// TIA Portal V20 export
// export: Created 2025-12-01T14:57:05.3623851Z, ExportSetting None, DisplayName Totally Integrated Automation Portal, DisplayVersion V20 Update 3, DisplayName TIA Portal Openness, DisplayVersion V20 Update 3, DisplayName TIA Portal Version Control Interface, DisplayVersion V20 Update 3, DisplayName STEP 7 Professional, DisplayVersion V20 Update 3, DisplayName STEP 7 Safety, DisplayVersion V20 Update 2, DisplayName WinCC Basic/Comfort/Advanced, DisplayVersion V20 Update 3, DisplayName WinCC Professional, DisplayVersion V20 Update 3, DisplayName WinCC Unified, DisplayVersion V20 Update 3
FUNCTION "FC776_Presion_DesPaletizador_Paletizador_Automatico" : Void   // FC776, STL
TITLE = Calculo de Presion del DesPaletizador
{ S7_Optimized_Access := 'FALSE' }
AUTHOR : TRACKING
NAME : 20130301
VERSION : 3.0
// stored: AutoNumber false
   VAR_INPUT
      Mesa : UInt;   // Mesa del DesPaletizador
      CalcularPresion : Bool;   // Orden de Calcular la Presion
   END_VAR
   VAR_IN_OUT
      PresionUT : Word;   // Presion ha utilizar para la UT de la Mesa
      FinCalculoPresion : Bool;   // Ya Realizado el Calculo de la Presion
   END_VAR
   VAR_TEMP
      NumeroUT : UInt;
   END_VAR
BEGIN

NETWORK
TITLE = Distribucion
////////////////////////////////////////////////////////////////////////////
// --- DISTRIBUCION
// ---

      AN    #FinCalculoPresion;
      A     #CalcularPresion;
      JC    CalcularDePresion;  // Calcular la Presion ?

      A     #FinCalculoPresion;
      AN    #CalcularPresion;
      JC    Fin_CalculoDePresion;  // Cierre de Protocolo ?

      BE;  // - Finalizar del Bloque



NETWORK
TITLE = Calcular la Presion
////////////////////////////////////////////////////////////////////////////
// --- CALCULAR LA PRESION
// ---
// --- Buscar la primera UT de la Mesa
// --- Recoger la Presion de la UT de la Base de Datos
// --- Dar por finalizado el Caculo, Activando el Protocolo
// ---

CalcularDePresion:NOP   0;
      L     "DB810_ColasMesas".Colas[#Mesa].UT_PrimeraMesa;
      T     #NumeroUT;

      SET;
      S     #FinCalculoPresion;  // Activar el Protocolo

// Presion para DesPaletizar y Paletizar
      L     "DB815_UTs_Datos".UT[#NumeroUT].Presion;
      T     #PresionUT;

      BE;  // - Finalizar del Bloque


////////////////////////////////////////////////////////////////////////////
// --- CIERRE DE PROTOCOLO
// ---

Fin_CalculoDePresion:NOP   0;

      SET;
      R     #FinCalculoPresion;  // - Cerrado el Protocolo
      L     0;
      T     #PresionUT;

      BE;  // - Finalizar del Bloque


END_FUNCTION
